// TIA Portal V20 export
DATA_BLOCK "Config"   // DB51
{ DB_Accessible_From_OPC_UA := 'FALSE' }
AUTHOR : ERsystem_FA2_DH. Kim
// stored: Access Published, DBAccessibleFromOPCUA false, DBAccessibleFromWebserver false, MemoryReserve 100, Namespace Unit1.Em5
   VAR RETAIN
      em { ExternalWritable := 'False'} : "LAF_typeEmConfiguration";
      axis { ExternalAccessible := 'False'; ExternalVisible := 'False'; ExternalWritable := 'False'} : Array[1.._.U1EM5_NO_OF_AXES] of DB_ANY;
      cam { ExternalAccessible := 'False'; ExternalVisible := 'False'; ExternalWritable := 'False'} : Array[1.._.U1EM5_NO_OF_CAM] of DB_ANY;
      outputCam { ExternalAccessible := 'False'; ExternalVisible := 'False'; ExternalWritable := 'False'} : Array[1.._.U1EM5_NO_OF_OUTPUTCAM] of DB_ANY;
      cmPnp1stCathodeDetect { S7_SetPoint := 'True'} : "LBC_typeDigitalSignalConfiguration";
      cmPnp2ndCathodeDetect { S7_SetPoint := 'True'} : "LBC_typeDigitalSignalConfiguration";
      cmCathodeAlignTableElectrodeDetect { S7_SetPoint := 'True'} : "LBC_typeDigitalSignalConfiguration";
      cmCathodeNgPnpElectrodeDetect { S7_SetPoint := 'True'} : "LBC_typeDigitalSignalConfiguration";
      cmCathodeNgBoxFullSensorDetect { S7_SetPoint := 'True'} : "LBC_typeDigitalSignalConfiguration";
      cmCathodeNgBoxDetect { S7_SetPoint := 'True'} : "LBC_typeDigitalSignalConfiguration";
      cmCathodeMainPnP1AxisX { ExternalAccessible := 'False'; ExternalVisible := 'False'; ExternalWritable := 'False'} : "LBC_typeAxis64PosConfiguration";
      cmCathodeMainPnP2AxisX { ExternalAccessible := 'False'; ExternalVisible := 'False'; ExternalWritable := 'False'} : "LBC_typeAxis64PosConfiguration";
      cmCathodeMainPnP1AxisY { ExternalAccessible := 'False'; ExternalVisible := 'False'; ExternalWritable := 'False'} : "LBC_typeAxis64PosConfiguration";
      cmCathodeMainPnP1AxisZ { ExternalAccessible := 'False'; ExternalVisible := 'False'; ExternalWritable := 'False'} : "LBC_typeAxis64PosConfiguration";
      cmCathodeMainPnP2AxisZ { ExternalAccessible := 'False'; ExternalVisible := 'False'; ExternalWritable := 'False'} : "LBC_typeAxis64PosConfiguration";
      cmCathodeAlignTableAxisX { ExternalAccessible := 'False'; ExternalVisible := 'False'; ExternalWritable := 'False'} : "LBC_typeAxis64PosConfiguration";
      cmCathodeAlignTableAxisY1 { ExternalAccessible := 'False'; ExternalVisible := 'False'; ExternalWritable := 'False'} : "LBC_typeAxis64PosConfiguration";
      cmCathodeAlignTableAxisY2 { ExternalAccessible := 'False'; ExternalVisible := 'False'; ExternalWritable := 'False'} : "LBC_typeAxis64PosConfiguration";
      cmCathodeMainPnP1RotaryCwCcw { ExternalAccessible := 'False'; ExternalVisible := 'False'; ExternalWritable := 'False'} : "LBC_typeTwoWayActuatorConfiguration";
      cmCathodeMainPnP1SuctionPlateVacuum { ExternalAccessible := 'False'; ExternalVisible := 'False'; ExternalWritable := 'False'} : "LBC_typeTwoWayActuatorConfiguration";
      cmCathodeMainPnP2SuctionPlateVacuum { ExternalAccessible := 'False'; ExternalVisible := 'False'; ExternalWritable := 'False'} : "LBC_typeTwoWayActuatorConfiguration";
      cmCathodeAlignTableSuctionPlateVacuum { ExternalAccessible := 'False'; ExternalVisible := 'False'; ExternalWritable := 'False'} : "LBC_typeTwoWayActuatorConfiguration";
      cmCathodeGlassCleaning { ExternalAccessible := 'False'; ExternalVisible := 'False'; ExternalWritable := 'False'} : "LBC_typeTwoWayActuatorConfiguration";
      cmCathodeNgPnpUpDown { ExternalAccessible := 'False'; ExternalVisible := 'False'; ExternalWritable := 'False'} : "LBC_typeTwoWayActuatorConfiguration";
      cmCathodeNgPnp1stFwdBwd { ExternalAccessible := 'False'; ExternalVisible := 'False'; ExternalWritable := 'False'; S7_SetPoint := 'True'} : "LBC_typeTwoWayActuatorConfiguration";
      cmCathodeNgPnp2ndFwdBwd { ExternalAccessible := 'False'; ExternalVisible := 'False'; ExternalWritable := 'False'; S7_SetPoint := 'True'} : "LBC_typeTwoWayActuatorConfiguration";
      cmCathodeMaintenanceMovingFixFrontRearFwdBwd { ExternalAccessible := 'False'; ExternalVisible := 'False'; ExternalWritable := 'False'} : "LBC_typeTwoWayActuatorConfiguration";
      cmCathodeNgBoxLiftUpDown { ExternalAccessible := 'False'; ExternalVisible := 'False'; ExternalWritable := 'False'; S7_SetPoint := 'True'} : "LBC_typeTwoWayActuatorConfiguration";
      cmCathodeNgBoxLockUpDown { ExternalAccessible := 'False'; ExternalVisible := 'False'; ExternalWritable := 'False'; S7_SetPoint := 'True'} : "LBC_typeTwoWayActuatorConfiguration";
      cmCathodeNgPnpVaccum { ExternalAccessible := 'False'; ExternalVisible := 'False'; ExternalWritable := 'False'; S7_SetPoint := 'True'} : "LBC_typeTwoWayActuatorConfiguration";
      cmCathodeConveyorCoverFwdBwd { S7_SetPoint := 'True'} : "LBC_typeTwoWayActuatorConfiguration";
      cmCathodeConveyorPickUpBlower { S7_SetPoint := 'True'} : "LBC_typeTwoWayActuatorConfiguration";
      cmCathodeVisionControllerInterface { ExternalAccessible := 'False'; ExternalVisible := 'False'; ExternalWritable := 'False'} : "LER_typeVisionConfiguration";
      softCam : Struct
         cmCathodeMainPnP1AxisX : "LER_typeSoftCamInterface";
         cmCathodeMainPnP2AxisX { S7_SetPoint := 'True'} : "LER_typeSoftCamInterface";
         cmCathodeMainPnP1AxisY { S7_SetPoint := 'True'} : "LER_typeSoftCamInterface";
         cmCathodeMainPnP1AxisZ { S7_SetPoint := 'True'} : "LER_typeSoftCamInterface";
         cmCathodeMainPnP2AxisZ { S7_SetPoint := 'True'} : "LER_typeSoftCamInterface";
         cmCathodeAlignTableAxisX { S7_SetPoint := 'True'} : "LER_typeSoftCamInterface";
         cmCathodeAlignTableAxisY1 { S7_SetPoint := 'True'} : "LER_typeSoftCamInterface";
         cmCathodeAlignTableAxisY2 { S7_SetPoint := 'True'} : "LER_typeSoftCamInterface";
      END_STRUCT;
   END_VAR
BEGIN
   em.referenceDesignator.parent := WSTRING#'';
   em.referenceDesignator.relative := WSTRING#'';
   em.referenceDesignator.combined := WSTRING#'';
   axis[1] := 146;   // CathodeMainPnP1AxisX
   axis[2] := 147;   // CathodeMainPnP2AxisX
   axis[3] := 152;   // CathodeMainPnP1AxisY
   axis[4] := 151;   // CathodeMainPnP1AxisZ
   axis[5] := 153;   // CathodeMainPnP2AxisZ
   axis[6] := 157;   // CathodeAlignTableAxisX
   axis[7] := 158;   // CathodeAlignTableAxisY1
   axis[8] := 159;   // CathodeAlignTableAxisY2
   cam[1] := 144;   // AnodeMainPnP1AxisX
   cam[2] := 145;   // AnodeMainPnP2AxisX
   cam[3] := 148;   // AnodeMainPnP1AxisY
   cam[4] := 149;   // AnodeMainPnP1AxisZ
   outputCam[1] := 416;
   outputCam[2] := 417;
   outputCam[3] := 419;
   outputCam[4] := 418;
   outputCam[5] := 422;
   outputCam[6] := 423;
   outputCam[7] := 428;
   outputCam[8] := 429;
   outputCam[9] := 421;
   outputCam[10] := 439;
   outputCam[11] := 427;
   outputCam[12] := 425;
   outputCam[13] := 457;
   outputCam[14] := 443;
   outputCam[15] := 424;
   outputCam[16] := 426;
   outputCam[17] := 444;
   outputCam[18] := 440;
   outputCam[19] := 458;
   cmPnp1stCathodeDetect.referenceDesignator := WSTRING#'DigitalSignal';
   cmPnp1stCathodeDetect.onDelay := T#0MS;
   cmPnp1stCathodeDetect.offDelay := T#0MS;
   cmPnp1stCathodeDetect.default := FALSE;
   cmPnp1stCathodeDetect.invertProcessValue := FALSE;
   cmPnp1stCathodeDetect.disableAlarms := FALSE;
   cmPnp2ndCathodeDetect.referenceDesignator := WSTRING#'DigitalSignal';
   cmPnp2ndCathodeDetect.onDelay := T#0MS;
   cmPnp2ndCathodeDetect.offDelay := T#0MS;
   cmPnp2ndCathodeDetect.default := FALSE;
   cmPnp2ndCathodeDetect.invertProcessValue := FALSE;
   cmPnp2ndCathodeDetect.disableAlarms := FALSE;
   cmCathodeAlignTableElectrodeDetect.referenceDesignator := WSTRING#'DigitalSignal';
   cmCathodeAlignTableElectrodeDetect.onDelay := T#0MS;
   cmCathodeAlignTableElectrodeDetect.offDelay := T#0MS;
   cmCathodeAlignTableElectrodeDetect.default := FALSE;
   cmCathodeAlignTableElectrodeDetect.invertProcessValue := FALSE;
   cmCathodeAlignTableElectrodeDetect.disableAlarms := FALSE;
   cmCathodeNgPnpElectrodeDetect.referenceDesignator := WSTRING#'DigitalSignal';
   cmCathodeNgPnpElectrodeDetect.onDelay := T#0MS;
   cmCathodeNgPnpElectrodeDetect.offDelay := T#0MS;
   cmCathodeNgPnpElectrodeDetect.default := FALSE;
   cmCathodeNgPnpElectrodeDetect.invertProcessValue := FALSE;
   cmCathodeNgPnpElectrodeDetect.disableAlarms := FALSE;
   cmCathodeNgBoxFullSensorDetect.referenceDesignator := WSTRING#'DigitalSignal';
   cmCathodeNgBoxFullSensorDetect.onDelay := T#0MS;
   cmCathodeNgBoxFullSensorDetect.offDelay := T#0MS;
   cmCathodeNgBoxFullSensorDetect.default := FALSE;
   cmCathodeNgBoxFullSensorDetect.invertProcessValue := FALSE;
   cmCathodeNgBoxFullSensorDetect.disableAlarms := FALSE;
   cmCathodeNgBoxDetect.referenceDesignator := WSTRING#'DigitalSignal';
   cmCathodeNgBoxDetect.onDelay := T#0MS;
   cmCathodeNgBoxDetect.offDelay := T#0MS;
   cmCathodeNgBoxDetect.default := FALSE;
   cmCathodeNgBoxDetect.invertProcessValue := FALSE;
   cmCathodeNgBoxDetect.disableAlarms := FALSE;
   cmCathodeMainPnP1AxisX.referenceDesignator := WSTRING#'CathodeMainPnP1AxisX';
   cmCathodeMainPnP1AxisX.disableAlarms := FALSE;
   cmCathodeMainPnP1AxisX.masterControlPopUp := TRUE;
   cmCathodeMainPnP1AxisX.setPositions[0].position := 0.0;
   cmCathodeMainPnP1AxisX.setPositions[1].position := 540.0;
   cmCathodeMainPnP1AxisX.setPositions[2].position := 544.0;
   cmCathodeMainPnP1AxisX.setPositions[3..15].position := 0.0;
   cmCathodeMainPnP1AxisX.setPositions[0..1].velocity := 500.0;
   cmCathodeMainPnP1AxisX.setPositions[2..3].velocity := 1040.0;
   cmCathodeMainPnP1AxisX.setPositions[4..15].velocity := -1.0;
   cmCathodeMainPnP1AxisX.setPositions[0..1].acceleration := 5000.0;
   cmCathodeMainPnP1AxisX.setPositions[2..3].acceleration := 10400.0;
   cmCathodeMainPnP1AxisX.setPositions[4..15].acceleration := -1.0;
   cmCathodeMainPnP1AxisX.setPositions[0..1].deceleration := 5000.0;
   cmCathodeMainPnP1AxisX.setPositions[2..3].deceleration := 10400.0;
   cmCathodeMainPnP1AxisX.setPositions[4..15].deceleration := -1.0;
   cmCathodeMainPnP1AxisX.setPositions[0..15]."name" := '';
   cmCathodeMainPnP2AxisX.referenceDesignator := WSTRING#'CathodeMainPnP2AxisX';
   cmCathodeMainPnP2AxisX.disableAlarms := FALSE;
   cmCathodeMainPnP2AxisX.masterControlPopUp := TRUE;
   cmCathodeMainPnP2AxisX.setPositions[0].position := 0.0;
   cmCathodeMainPnP2AxisX.setPositions[1].position := 540.0;
   cmCathodeMainPnP2AxisX.setPositions[2].position := 538.0;
   cmCathodeMainPnP2AxisX.setPositions[3..15].position := 0.0;
   cmCathodeMainPnP2AxisX.setPositions[0..1].velocity := 500.0;
   cmCathodeMainPnP2AxisX.setPositions[2..3].velocity := 1040.0;
   cmCathodeMainPnP2AxisX.setPositions[4..15].velocity := -1.0;
   cmCathodeMainPnP2AxisX.setPositions[0..1].acceleration := 5000.0;
   cmCathodeMainPnP2AxisX.setPositions[2..3].acceleration := 10400.0;
   cmCathodeMainPnP2AxisX.setPositions[4..15].acceleration := -1.0;
   cmCathodeMainPnP2AxisX.setPositions[0..1].deceleration := 5000.0;
   cmCathodeMainPnP2AxisX.setPositions[2..3].deceleration := 10400.0;
   cmCathodeMainPnP2AxisX.setPositions[4..15].deceleration := -1.0;
   cmCathodeMainPnP2AxisX.setPositions[0..15]."name" := '';
   cmCathodeMainPnP1AxisY.referenceDesignator := WSTRING#'CathodeMainPnP1AxisY';
   cmCathodeMainPnP1AxisY.disableAlarms := FALSE;
   cmCathodeMainPnP1AxisY.masterControlPopUp := TRUE;
   cmCathodeMainPnP1AxisY.setPositions[0..15].position := 0.0;
   cmCathodeMainPnP1AxisY.setPositions[0].velocity := 50.0;
   cmCathodeMainPnP1AxisY.setPositions[1].velocity := 30.0;
   cmCathodeMainPnP1AxisY.setPositions[2..15].velocity := -1.0;
   cmCathodeMainPnP1AxisY.setPositions[0].acceleration := 500.0;
   cmCathodeMainPnP1AxisY.setPositions[1].acceleration := 30.0;
   cmCathodeMainPnP1AxisY.setPositions[2..15].acceleration := -1.0;
   cmCathodeMainPnP1AxisY.setPositions[0].deceleration := 500.0;
   cmCathodeMainPnP1AxisY.setPositions[1].deceleration := 30.0;
   cmCathodeMainPnP1AxisY.setPositions[2..15].deceleration := -1.0;
   cmCathodeMainPnP1AxisY.setPositions[0..15]."name" := '';
   cmCathodeMainPnP1AxisZ.referenceDesignator := WSTRING#'CathodeMainPnP1AxisZ';
   cmCathodeMainPnP1AxisZ.disableAlarms := FALSE;
   cmCathodeMainPnP1AxisZ.masterControlPopUp := TRUE;
   cmCathodeMainPnP1AxisZ.setPositions[0].position := 0.0;
   cmCathodeMainPnP1AxisZ.setPositions[1].position := 20.0;
   cmCathodeMainPnP1AxisZ.setPositions[2].position := 30.0;
   cmCathodeMainPnP1AxisZ.setPositions[3..15].position := 0.0;
   cmCathodeMainPnP1AxisZ.setPositions[0..3].velocity := 50.0;
   cmCathodeMainPnP1AxisZ.setPositions[4..15].velocity := -1.0;
   cmCathodeMainPnP1AxisZ.setPositions[0..3].acceleration := 500.0;
   cmCathodeMainPnP1AxisZ.setPositions[4..15].acceleration := -1.0;
   cmCathodeMainPnP1AxisZ.setPositions[0..3].deceleration := 500.0;
   cmCathodeMainPnP1AxisZ.setPositions[4..15].deceleration := -1.0;
   cmCathodeMainPnP1AxisZ.setPositions[0..15]."name" := '';
   cmCathodeMainPnP2AxisZ.referenceDesignator := WSTRING#'CathodeMainPnP2AxisZ';
   cmCathodeMainPnP2AxisZ.disableAlarms := FALSE;
   cmCathodeMainPnP2AxisZ.masterControlPopUp := TRUE;
   cmCathodeMainPnP2AxisZ.setPositions[0].position := 0.0;
   cmCathodeMainPnP2AxisZ.setPositions[1].position := 20.0;
   cmCathodeMainPnP2AxisZ.setPositions[2].position := 30.0;
   cmCathodeMainPnP2AxisZ.setPositions[3..15].position := 0.0;
   cmCathodeMainPnP2AxisZ.setPositions[0..3].velocity := 50.0;
   cmCathodeMainPnP2AxisZ.setPositions[4..15].velocity := -1.0;
   cmCathodeMainPnP2AxisZ.setPositions[0..3].acceleration := 500.0;
   cmCathodeMainPnP2AxisZ.setPositions[4..15].acceleration := -1.0;
   cmCathodeMainPnP2AxisZ.setPositions[0..3].deceleration := 500.0;
   cmCathodeMainPnP2AxisZ.setPositions[4..15].deceleration := -1.0;
   cmCathodeMainPnP2AxisZ.setPositions[0..15]."name" := '';
   cmCathodeAlignTableAxisX.referenceDesignator := WSTRING#'CathodeAlignTableAxisX';
   cmCathodeAlignTableAxisX.disableAlarms := FALSE;
   cmCathodeAlignTableAxisX.masterControlPopUp := TRUE;
   cmCathodeAlignTableAxisX.setPositions[0].position := 0.0;
   cmCathodeAlignTableAxisX.setPositions[1].position := 1.0;
   cmCathodeAlignTableAxisX.setPositions[2..3].position := 1.07;
   cmCathodeAlignTableAxisX.setPositions[4].position := -0.93;
   cmCathodeAlignTableAxisX.setPositions[5..7].position := -2.93;
   cmCathodeAlignTableAxisX.setPositions[8].position := -0.93;
   cmCathodeAlignTableAxisX.setPositions[9].position := 1.07;
   cmCathodeAlignTableAxisX.setPositions[10..15].position := 0.0;
   cmCathodeAlignTableAxisX.setPositions[0..1].velocity := 50.0;
   cmCathodeAlignTableAxisX.setPositions[2..9].velocity := 30.0;
   cmCathodeAlignTableAxisX.setPositions[10..15].velocity := -1.0;
   cmCathodeAlignTableAxisX.setPositions[0..1].acceleration := 500.0;
   cmCathodeAlignTableAxisX.setPositions[2..9].acceleration := 30.0;
   cmCathodeAlignTableAxisX.setPositions[10..15].acceleration := -1.0;
   cmCathodeAlignTableAxisX.setPositions[0..1].deceleration := 500.0;
   cmCathodeAlignTableAxisX.setPositions[2..9].deceleration := 30.0;
   cmCathodeAlignTableAxisX.setPositions[10..15].deceleration := -1.0;
   cmCathodeAlignTableAxisX.setPositions[0..15]."name" := '';
   cmCathodeAlignTableAxisY1.referenceDesignator := WSTRING#'CathodeAlignTableAxisY1';
   cmCathodeAlignTableAxisY1.disableAlarms := FALSE;
   cmCathodeAlignTableAxisY1.masterControlPopUp := TRUE;
   cmCathodeAlignTableAxisY1.setPositions[0].position := 0.0;
   cmCathodeAlignTableAxisY1.setPositions[1].position := 2.0;
   cmCathodeAlignTableAxisY1.setPositions[2].position := 0.15;
   cmCathodeAlignTableAxisY1.setPositions[3..5].position := 2.15;
   cmCathodeAlignTableAxisY1.setPositions[6].position := 0.15;
   cmCathodeAlignTableAxisY1.setPositions[7].position := -1.85;
   cmCathodeAlignTableAxisY1.setPositions[8].position := 0.15;
   cmCathodeAlignTableAxisY1.setPositions[9].position := -1.85;
   cmCathodeAlignTableAxisY1.setPositions[10..15].position := 0.0;
   cmCathodeAlignTableAxisY1.setPositions[0..1].velocity := 50.0;
   cmCathodeAlignTableAxisY1.setPositions[2..9].velocity := 30.0;
   cmCathodeAlignTableAxisY1.setPositions[10..15].velocity := -1.0;
   cmCathodeAlignTableAxisY1.setPositions[0..1].acceleration := 500.0;
   cmCathodeAlignTableAxisY1.setPositions[2..9].acceleration := 30.0;
   cmCathodeAlignTableAxisY1.setPositions[10..15].acceleration := -1.0;
   cmCathodeAlignTableAxisY1.setPositions[0..1].deceleration := 500.0;
   cmCathodeAlignTableAxisY1.setPositions[2..9].deceleration := 30.0;
   cmCathodeAlignTableAxisY1.setPositions[10..15].deceleration := -1.0;
   cmCathodeAlignTableAxisY1.setPositions[0..15]."name" := '';
   cmCathodeAlignTableAxisY2.referenceDesignator := WSTRING#'CathodeAlignTableAxisY2';
   cmCathodeAlignTableAxisY2.disableAlarms := FALSE;
   cmCathodeAlignTableAxisY2.masterControlPopUp := TRUE;
   cmCathodeAlignTableAxisY2.setPositions[0].position := 0.0;
   cmCathodeAlignTableAxisY2.setPositions[1].position := 3.0;
   cmCathodeAlignTableAxisY2.setPositions[2].position := -0.96;
   cmCathodeAlignTableAxisY2.setPositions[3..5].position := -2.96;
   cmCathodeAlignTableAxisY2.setPositions[6].position := -0.96;
   cmCathodeAlignTableAxisY2.setPositions[7].position := 1.04;
   cmCathodeAlignTableAxisY2.setPositions[8].position := -0.96;
   cmCathodeAlignTableAxisY2.setPositions[9].position := 1.04;
   cmCathodeAlignTableAxisY2.setPositions[10..15].position := 0.0;
   cmCathodeAlignTableAxisY2.setPositions[0..1].velocity := 50.0;
   cmCathodeAlignTableAxisY2.setPositions[2..9].velocity := 30.0;
   cmCathodeAlignTableAxisY2.setPositions[10..15].velocity := -1.0;
   cmCathodeAlignTableAxisY2.setPositions[0..1].acceleration := 500.0;
   cmCathodeAlignTableAxisY2.setPositions[2..9].acceleration := 30.0;
   cmCathodeAlignTableAxisY2.setPositions[10..15].acceleration := -1.0;
   cmCathodeAlignTableAxisY2.setPositions[0..1].deceleration := 500.0;
   cmCathodeAlignTableAxisY2.setPositions[2..9].deceleration := 30.0;
   cmCathodeAlignTableAxisY2.setPositions[10..15].deceleration := -1.0;
   cmCathodeAlignTableAxisY2.setPositions[0..15]."name" := '';
   cmCathodeMainPnP1RotaryCwCcw.referenceDesignator := WSTRING#'MainPnP1RotaryCwCcw';
   cmCathodeMainPnP1RotaryCwCcw.monitoringLeavingFeedback := T#1S;
   cmCathodeMainPnP1RotaryCwCcw.monitoringReachingFeedback := T#1S;
   cmCathodeMainPnP1RotaryCwCcw.monitoringDiscrepancy := T#0MS;
   cmCathodeMainPnP1RotaryCwCcw.setOutputHomeContinuously := TRUE;
   cmCathodeMainPnP1RotaryCwCcw.setOutputWorkContinuously := TRUE;
   cmCathodeMainPnP1RotaryCwCcw.disableHomeCommand := FALSE;
   cmCathodeMainPnP1RotaryCwCcw.disableFeedbackHomePos := FALSE;
   cmCathodeMainPnP1RotaryCwCcw.disableFeedbackWorkPos := FALSE;
   cmCathodeMainPnP1RotaryCwCcw.disableAlarms := TRUE;
   cmCathodeMainPnP1RotaryCwCcw.resetOutputsOnError := FALSE;
   cmCathodeMainPnP1RotaryCwCcw.allwaysWaitOnReachingTime := FALSE;
   cmCathodeMainPnP1SuctionPlateVacuum.referenceDesignator := WSTRING#'MainPnP1Vacuum';
   cmCathodeMainPnP1SuctionPlateVacuum.monitoringLeavingFeedback := T#1S;
   cmCathodeMainPnP1SuctionPlateVacuum.monitoringReachingFeedback := T#1S;
   cmCathodeMainPnP1SuctionPlateVacuum.monitoringDiscrepancy := T#15S;
   cmCathodeMainPnP1SuctionPlateVacuum.setOutputHomeContinuously := TRUE;
   cmCathodeMainPnP1SuctionPlateVacuum.setOutputWorkContinuously := TRUE;
   cmCathodeMainPnP1SuctionPlateVacuum.disableHomeCommand := FALSE;
   cmCathodeMainPnP1SuctionPlateVacuum.disableFeedbackHomePos := FALSE;
   cmCathodeMainPnP1SuctionPlateVacuum.disableFeedbackWorkPos := FALSE;
   cmCathodeMainPnP1SuctionPlateVacuum.disableAlarms := FALSE;
   cmCathodeMainPnP1SuctionPlateVacuum.resetOutputsOnError := FALSE;
   cmCathodeMainPnP1SuctionPlateVacuum.allwaysWaitOnReachingTime := FALSE;
   cmCathodeMainPnP2SuctionPlateVacuum.referenceDesignator := WSTRING#'MainPnP2Vacuum';
   cmCathodeMainPnP2SuctionPlateVacuum.monitoringLeavingFeedback := T#1S;
   cmCathodeMainPnP2SuctionPlateVacuum.monitoringReachingFeedback := T#1S;
   cmCathodeMainPnP2SuctionPlateVacuum.monitoringDiscrepancy := T#15S;
   cmCathodeMainPnP2SuctionPlateVacuum.setOutputHomeContinuously := TRUE;
   cmCathodeMainPnP2SuctionPlateVacuum.setOutputWorkContinuously := TRUE;
   cmCathodeMainPnP2SuctionPlateVacuum.disableHomeCommand := FALSE;
   cmCathodeMainPnP2SuctionPlateVacuum.disableFeedbackHomePos := FALSE;
   cmCathodeMainPnP2SuctionPlateVacuum.disableFeedbackWorkPos := FALSE;
   cmCathodeMainPnP2SuctionPlateVacuum.disableAlarms := FALSE;
   cmCathodeMainPnP2SuctionPlateVacuum.resetOutputsOnError := FALSE;
   cmCathodeMainPnP2SuctionPlateVacuum.allwaysWaitOnReachingTime := FALSE;
   cmCathodeAlignTableSuctionPlateVacuum.referenceDesignator := WSTRING#'AlignTableVaccum';
   cmCathodeAlignTableSuctionPlateVacuum.monitoringLeavingFeedback := T#1S;
   cmCathodeAlignTableSuctionPlateVacuum.monitoringReachingFeedback := T#1S;
   cmCathodeAlignTableSuctionPlateVacuum.monitoringDiscrepancy := T#0MS;
   cmCathodeAlignTableSuctionPlateVacuum.setOutputHomeContinuously := TRUE;
   cmCathodeAlignTableSuctionPlateVacuum.setOutputWorkContinuously := TRUE;
   cmCathodeAlignTableSuctionPlateVacuum.disableHomeCommand := FALSE;
   cmCathodeAlignTableSuctionPlateVacuum.disableFeedbackHomePos := FALSE;
   cmCathodeAlignTableSuctionPlateVacuum.disableFeedbackWorkPos := FALSE;
   cmCathodeAlignTableSuctionPlateVacuum.disableAlarms := FALSE;
   cmCathodeAlignTableSuctionPlateVacuum.resetOutputsOnError := FALSE;
   cmCathodeAlignTableSuctionPlateVacuum.allwaysWaitOnReachingTime := FALSE;
   cmCathodeGlassCleaning.referenceDesignator := WSTRING#'GlassCleaning';
   cmCathodeGlassCleaning.monitoringLeavingFeedback := T#1S;
   cmCathodeGlassCleaning.monitoringReachingFeedback := T#1S;
   cmCathodeGlassCleaning.monitoringDiscrepancy := T#0MS;
   cmCathodeGlassCleaning.setOutputHomeContinuously := TRUE;
   cmCathodeGlassCleaning.setOutputWorkContinuously := TRUE;
   cmCathodeGlassCleaning.disableHomeCommand := FALSE;
   cmCathodeGlassCleaning.disableFeedbackHomePos := TRUE;
   cmCathodeGlassCleaning.disableFeedbackWorkPos := TRUE;
   cmCathodeGlassCleaning.disableAlarms := TRUE;
   cmCathodeGlassCleaning.resetOutputsOnError := FALSE;
   cmCathodeGlassCleaning.allwaysWaitOnReachingTime := FALSE;
   cmCathodeNgPnpUpDown.referenceDesignator := WSTRING#'NgPnpUpDown';
   cmCathodeNgPnpUpDown.monitoringLeavingFeedback := T#5S;
   cmCathodeNgPnpUpDown.monitoringReachingFeedback := T#5S;
   cmCathodeNgPnpUpDown.monitoringDiscrepancy := T#0MS;
   cmCathodeNgPnpUpDown.setOutputHomeContinuously := TRUE;
   cmCathodeNgPnpUpDown.setOutputWorkContinuously := TRUE;
   cmCathodeNgPnpUpDown.disableHomeCommand := FALSE;
   cmCathodeNgPnpUpDown.disableFeedbackHomePos := TRUE;
   cmCathodeNgPnpUpDown.disableFeedbackWorkPos := TRUE;
   cmCathodeNgPnpUpDown.disableAlarms := FALSE;
   cmCathodeNgPnpUpDown.resetOutputsOnError := FALSE;
   cmCathodeNgPnpUpDown.allwaysWaitOnReachingTime := FALSE;
   cmCathodeNgPnp1stFwdBwd.referenceDesignator := WSTRING#'NgPnp1stFwdBwd';
   cmCathodeNgPnp1stFwdBwd.monitoringLeavingFeedback := T#5S;
   cmCathodeNgPnp1stFwdBwd.monitoringReachingFeedback := T#5S;
   cmCathodeNgPnp1stFwdBwd.monitoringDiscrepancy := T#0MS;
   cmCathodeNgPnp1stFwdBwd.setOutputHomeContinuously := TRUE;
   cmCathodeNgPnp1stFwdBwd.setOutputWorkContinuously := TRUE;
   cmCathodeNgPnp1stFwdBwd.disableHomeCommand := FALSE;
   cmCathodeNgPnp1stFwdBwd.disableFeedbackHomePos := FALSE;
   cmCathodeNgPnp1stFwdBwd.disableFeedbackWorkPos := FALSE;
   cmCathodeNgPnp1stFwdBwd.disableAlarms := FALSE;
   cmCathodeNgPnp1stFwdBwd.resetOutputsOnError := FALSE;
   cmCathodeNgPnp1stFwdBwd.allwaysWaitOnReachingTime := FALSE;
   cmCathodeNgPnp2ndFwdBwd.referenceDesignator := WSTRING#'NgPnp2ndFwdBwd';
   cmCathodeNgPnp2ndFwdBwd.monitoringLeavingFeedback := T#5S;
   cmCathodeNgPnp2ndFwdBwd.monitoringReachingFeedback := T#5S;
   cmCathodeNgPnp2ndFwdBwd.monitoringDiscrepancy := T#0MS;
   cmCathodeNgPnp2ndFwdBwd.setOutputHomeContinuously := TRUE;
   cmCathodeNgPnp2ndFwdBwd.setOutputWorkContinuously := TRUE;
   cmCathodeNgPnp2ndFwdBwd.disableHomeCommand := FALSE;
   cmCathodeNgPnp2ndFwdBwd.disableFeedbackHomePos := TRUE;
   cmCathodeNgPnp2ndFwdBwd.disableFeedbackWorkPos := TRUE;
   cmCathodeNgPnp2ndFwdBwd.disableAlarms := FALSE;
   cmCathodeNgPnp2ndFwdBwd.resetOutputsOnError := FALSE;
   cmCathodeNgPnp2ndFwdBwd.allwaysWaitOnReachingTime := FALSE;
   cmCathodeMaintenanceMovingFixFrontRearFwdBwd.referenceDesignator := WSTRING#'MaintenanceFix';
   cmCathodeMaintenanceMovingFixFrontRearFwdBwd.monitoringLeavingFeedback := T#5S;
   cmCathodeMaintenanceMovingFixFrontRearFwdBwd.monitoringReachingFeedback := T#5S;
   cmCathodeMaintenanceMovingFixFrontRearFwdBwd.monitoringDiscrepancy := T#0MS;
   cmCathodeMaintenanceMovingFixFrontRearFwdBwd.setOutputHomeContinuously := TRUE;
   cmCathodeMaintenanceMovingFixFrontRearFwdBwd.setOutputWorkContinuously := TRUE;
   cmCathodeMaintenanceMovingFixFrontRearFwdBwd.disableHomeCommand := FALSE;
   cmCathodeMaintenanceMovingFixFrontRearFwdBwd.disableFeedbackHomePos := FALSE;
   cmCathodeMaintenanceMovingFixFrontRearFwdBwd.disableFeedbackWorkPos := FALSE;
   cmCathodeMaintenanceMovingFixFrontRearFwdBwd.disableAlarms := FALSE;
   cmCathodeMaintenanceMovingFixFrontRearFwdBwd.resetOutputsOnError := FALSE;
   cmCathodeMaintenanceMovingFixFrontRearFwdBwd.allwaysWaitOnReachingTime := FALSE;
   cmCathodeNgBoxLiftUpDown.referenceDesignator := WSTRING#'NgBoxLiftUpDown';
   cmCathodeNgBoxLiftUpDown.monitoringLeavingFeedback := T#5S;
   cmCathodeNgBoxLiftUpDown.monitoringReachingFeedback := T#5S;
   cmCathodeNgBoxLiftUpDown.monitoringDiscrepancy := T#0MS;
   cmCathodeNgBoxLiftUpDown.setOutputHomeContinuously := TRUE;
   cmCathodeNgBoxLiftUpDown.setOutputWorkContinuously := TRUE;
   cmCathodeNgBoxLiftUpDown.disableHomeCommand := FALSE;
   cmCathodeNgBoxLiftUpDown.disableFeedbackHomePos := FALSE;
   cmCathodeNgBoxLiftUpDown.disableFeedbackWorkPos := FALSE;
   cmCathodeNgBoxLiftUpDown.disableAlarms := FALSE;
   cmCathodeNgBoxLiftUpDown.resetOutputsOnError := FALSE;
   cmCathodeNgBoxLiftUpDown.allwaysWaitOnReachingTime := FALSE;
   cmCathodeNgBoxLockUpDown.referenceDesignator := WSTRING#'NgBoxLockUpDown';
   cmCathodeNgBoxLockUpDown.monitoringLeavingFeedback := T#5S;
   cmCathodeNgBoxLockUpDown.monitoringReachingFeedback := T#5S;
   cmCathodeNgBoxLockUpDown.monitoringDiscrepancy := T#0MS;
   cmCathodeNgBoxLockUpDown.setOutputHomeContinuously := TRUE;
   cmCathodeNgBoxLockUpDown.setOutputWorkContinuously := TRUE;
   cmCathodeNgBoxLockUpDown.disableHomeCommand := FALSE;
   cmCathodeNgBoxLockUpDown.disableFeedbackHomePos := FALSE;
   cmCathodeNgBoxLockUpDown.disableFeedbackWorkPos := FALSE;
   cmCathodeNgBoxLockUpDown.disableAlarms := FALSE;
   cmCathodeNgBoxLockUpDown.resetOutputsOnError := FALSE;
   cmCathodeNgBoxLockUpDown.allwaysWaitOnReachingTime := FALSE;
   cmCathodeNgPnpVaccum.referenceDesignator := WSTRING#'NgPnpVaccum';
   cmCathodeNgPnpVaccum.monitoringLeavingFeedback := T#5S;
   cmCathodeNgPnpVaccum.monitoringReachingFeedback := T#5S;
   cmCathodeNgPnpVaccum.monitoringDiscrepancy := T#0MS;
   cmCathodeNgPnpVaccum.setOutputHomeContinuously := TRUE;
   cmCathodeNgPnpVaccum.setOutputWorkContinuously := TRUE;
   cmCathodeNgPnpVaccum.disableHomeCommand := FALSE;
   cmCathodeNgPnpVaccum.disableFeedbackHomePos := FALSE;
   cmCathodeNgPnpVaccum.disableFeedbackWorkPos := FALSE;
   cmCathodeNgPnpVaccum.disableAlarms := FALSE;
   cmCathodeNgPnpVaccum.resetOutputsOnError := FALSE;
   cmCathodeNgPnpVaccum.allwaysWaitOnReachingTime := FALSE;
   cmCathodeConveyorCoverFwdBwd.referenceDesignator := WSTRING#'ConveyorCoverFwdBwd';
   cmCathodeConveyorCoverFwdBwd.monitoringLeavingFeedback := T#5S;
   cmCathodeConveyorCoverFwdBwd.monitoringReachingFeedback := T#5S;
   cmCathodeConveyorCoverFwdBwd.monitoringDiscrepancy := T#0MS;
   cmCathodeConveyorCoverFwdBwd.setOutputHomeContinuously := TRUE;
   cmCathodeConveyorCoverFwdBwd.setOutputWorkContinuously := TRUE;
   cmCathodeConveyorCoverFwdBwd.disableHomeCommand := FALSE;
   cmCathodeConveyorCoverFwdBwd.disableFeedbackHomePos := TRUE;
   cmCathodeConveyorCoverFwdBwd.disableFeedbackWorkPos := TRUE;
   cmCathodeConveyorCoverFwdBwd.disableAlarms := FALSE;
   cmCathodeConveyorCoverFwdBwd.resetOutputsOnError := FALSE;
   cmCathodeConveyorCoverFwdBwd.allwaysWaitOnReachingTime := FALSE;
   cmCathodeConveyorPickUpBlower.referenceDesignator := WSTRING#'ConveyorPickUpBlower';
   cmCathodeConveyorPickUpBlower.monitoringLeavingFeedback := T#0MS;
   cmCathodeConveyorPickUpBlower.monitoringReachingFeedback := T#0MS;
   cmCathodeConveyorPickUpBlower.monitoringDiscrepancy := T#0MS;
   cmCathodeConveyorPickUpBlower.setOutputHomeContinuously := TRUE;
   cmCathodeConveyorPickUpBlower.setOutputWorkContinuously := TRUE;
   cmCathodeConveyorPickUpBlower.disableHomeCommand := FALSE;
   cmCathodeConveyorPickUpBlower.disableFeedbackHomePos := TRUE;
   cmCathodeConveyorPickUpBlower.disableFeedbackWorkPos := TRUE;
   cmCathodeConveyorPickUpBlower.disableAlarms := FALSE;
   cmCathodeConveyorPickUpBlower.resetOutputsOnError := FALSE;
   cmCathodeConveyorPickUpBlower.allwaysWaitOnReachingTime := FALSE;
   cmCathodeVisionControllerInterface.hwID.cmdResultStatusID := 770;
   cmCathodeVisionControllerInterface.hwID.trgReadyStatusID := 771;
   cmCathodeVisionControllerInterface.hwID.trgAckStatusID := 772;
   cmCathodeVisionControllerInterface.hwID.miscellaneousStatusID := 773;
   cmCathodeVisionControllerInterface.hwID.assignableStatusID := 774;
   cmCathodeVisionControllerInterface.hwID.resultData248ByteID_1 := 791;
   cmCathodeVisionControllerInterface.hwID.resultData248ByteID_2 := 984;
   cmCathodeVisionControllerInterface.hwID.resultData248ByteID_3 := 987;
   cmCathodeVisionControllerInterface.hwID.resultData248ByteID_4 := 988;
   cmCathodeVisionControllerInterface.hwID.resultData248ByteID_5 := 989;
   cmCathodeVisionControllerInterface.hwID.cmdResultControlID := 940;
   cmCathodeVisionControllerInterface.hwID.trgControlID := 941;
   cmCathodeVisionControllerInterface.hwID.miscellaneousControlID := 942;
   cmCathodeVisionControllerInterface.hwID.reservedControlID := 943;
   cmCathodeVisionControllerInterface.hwID.assignableControlID := 944;
   cmCathodeVisionControllerInterface.hwID.parameterData248ByteID_1 := 945;
   cmCathodeVisionControllerInterface.hwID.parameterData248ByteID_2 := 990;
   cmCathodeVisionControllerInterface.hwID.parameterData248ByteID_3 := 991;
   cmCathodeVisionControllerInterface.hwID.parameterData248ByteID_4 := 992;
   cmCathodeVisionControllerInterface.hwID.parameterData248ByteID_5 := 993;
   cmCathodeVisionControllerInterface.referenceDesignator := WSTRING#'';
   cmCathodeVisionControllerInterface.disableAlarms := FALSE;
   cmCathodeVisionControllerInterface.trigger1Use := FALSE;
   cmCathodeVisionControllerInterface.trigger2Use := FALSE;
   cmCathodeVisionControllerInterface.trigger3Use := FALSE;
   cmCathodeVisionControllerInterface.trigger4Use := FALSE;
   cmCathodeVisionControllerInterface.triggertime := T#0MS;
   cmCathodeVisionControllerInterface.cycleTime := T#0MS;
   cmCathodeVisionControllerInterface.DataConfig.cmdResultControl.cmdRequest := FALSE;
   cmCathodeVisionControllerInterface.DataConfig.cmdResultControl.inDataFbSyncInhibit := FALSE;
   cmCathodeVisionControllerInterface.DataConfig.cmdResultControl.reserved := FALSE;
   cmCathodeVisionControllerInterface.DataConfig.cmdResultControl.resultAck := FALSE;
   cmCathodeVisionControllerInterface.DataConfig.cmdResultControl.err0ResetRequest := FALSE;
   cmCathodeVisionControllerInterface.DataConfig.cmdResultControl.err1ResetRequest := FALSE;
   cmCathodeVisionControllerInterface.DataConfig.cmdResultControl.reserved0 := FALSE;
   cmCathodeVisionControllerInterface.DataConfig.cmdResultControl.reserved1 := FALSE;
   cmCathodeVisionControllerInterface.DataConfig.trgControl.trg1 := FALSE;
   cmCathodeVisionControllerInterface.DataConfig.trgControl.trg2 := FALSE;
   cmCathodeVisionControllerInterface.DataConfig.trgControl.trg3 := FALSE;
   cmCathodeVisionControllerInterface.DataConfig.trgControl.trg4 := FALSE;
   cmCathodeVisionControllerInterface.DataConfig.trgControl.reserved0 := FALSE;
   cmCathodeVisionControllerInterface.DataConfig.trgControl.reserved1 := FALSE;
   cmCathodeVisionControllerInterface.DataConfig.trgControl.reserved2 := FALSE;
   cmCathodeVisionControllerInterface.DataConfig.trgControl.reserved3 := FALSE;
   cmCathodeVisionControllerInterface.DataConfig.miscellaneousControl.reset := FALSE;
   cmCathodeVisionControllerInterface.DataConfig.miscellaneousControl.ext := FALSE;
   cmCathodeVisionControllerInterface.DataConfig.miscellaneousControl.test := FALSE;
   cmCathodeVisionControllerInterface.DataConfig.miscellaneousControl.reserved0 := FALSE;
   cmCathodeVisionControllerInterface.DataConfig.miscellaneousControl.reserved1 := FALSE;
   cmCathodeVisionControllerInterface.DataConfig.miscellaneousControl.reserved2 := FALSE;
   cmCathodeVisionControllerInterface.DataConfig.miscellaneousControl.reserved3 := FALSE;
   cmCathodeVisionControllerInterface.DataConfig.miscellaneousControl.reserved4 := FALSE;
   cmCathodeVisionControllerInterface.DataConfig.reservedControl.reserved0 := FALSE;
   cmCathodeVisionControllerInterface.DataConfig.reservedControl.reserved1 := FALSE;
   cmCathodeVisionControllerInterface.DataConfig.reservedControl.reserved2 := FALSE;
   cmCathodeVisionControllerInterface.DataConfig.reservedControl.reserved3 := FALSE;
   cmCathodeVisionControllerInterface.DataConfig.reservedControl.reserved4 := FALSE;
   cmCathodeVisionControllerInterface.DataConfig.reservedControl.reserved5 := FALSE;
   cmCathodeVisionControllerInterface.DataConfig.reservedControl.reserved6 := FALSE;
   cmCathodeVisionControllerInterface.DataConfig.reservedControl.reserved7 := FALSE;
   cmCathodeVisionControllerInterface.DataConfig.assignableControl.assignable_0 := FALSE;
   cmCathodeVisionControllerInterface.DataConfig.assignableControl.assignable_1 := FALSE;
   cmCathodeVisionControllerInterface.DataConfig.assignableControl.assignable_2 := FALSE;
   cmCathodeVisionControllerInterface.DataConfig.assignableControl.assignable_3 := FALSE;
   cmCathodeVisionControllerInterface.DataConfig.assignableControl.assignable_4 := FALSE;
   cmCathodeVisionControllerInterface.DataConfig.assignableControl.assignable_5 := FALSE;
   cmCathodeVisionControllerInterface.DataConfig.assignableControl.assignable_6 := FALSE;
   cmCathodeVisionControllerInterface.DataConfig.assignableControl.assignable_7 := FALSE;
   cmCathodeVisionControllerInterface.DataConfig.assignableControl.assignable_8 := FALSE;
   cmCathodeVisionControllerInterface.DataConfig.assignableControl.assignable_9 := FALSE;
   cmCathodeVisionControllerInterface.DataConfig.assignableControl.assignable_10 := FALSE;
   cmCathodeVisionControllerInterface.DataConfig.assignableControl.assignable_11 := FALSE;
   cmCathodeVisionControllerInterface.DataConfig.assignableControl.assignable_12 := FALSE;
   cmCathodeVisionControllerInterface.DataConfig.assignableControl.assignable_13 := FALSE;
   cmCathodeVisionControllerInterface.DataConfig.assignableControl.assignable_14 := FALSE;
   cmCathodeVisionControllerInterface.DataConfig.assignableControl.assignable_15 := FALSE;
   cmCathodeVisionControllerInterface.DataConfig.assignableControl.assignable_16 := FALSE;
   cmCathodeVisionControllerInterface.DataConfig.assignableControl.assignable_17 := FALSE;
   cmCathodeVisionControllerInterface.DataConfig.assignableControl.assignable_18 := FALSE;
   cmCathodeVisionControllerInterface.DataConfig.assignableControl.assignable_19 := FALSE;
   cmCathodeVisionControllerInterface.DataConfig.assignableControl.assignable_20 := FALSE;
   cmCathodeVisionControllerInterface.DataConfig.assignableControl.assignable_21 := FALSE;
   cmCathodeVisionControllerInterface.DataConfig.assignableControl.assignable_22 := FALSE;
   cmCathodeVisionControllerInterface.DataConfig.assignableControl.assignable_23 := FALSE;
   cmCathodeVisionControllerInterface.DataConfig.assignableControl.assignable_24 := FALSE;
   cmCathodeVisionControllerInterface.DataConfig.assignableControl.assignable_25 := FALSE;
   cmCathodeVisionControllerInterface.DataConfig.assignableControl.assignable_26 := FALSE;
   cmCathodeVisionControllerInterface.DataConfig.assignableControl.assignable_27 := FALSE;
   cmCathodeVisionControllerInterface.DataConfig.assignableControl.assignable_28 := FALSE;
   cmCathodeVisionControllerInterface.DataConfig.assignableControl.assignable_29 := FALSE;
   cmCathodeVisionControllerInterface.DataConfig.assignableControl.assignable_30 := FALSE;
   cmCathodeVisionControllerInterface.DataConfig.assignableControl.assignable_31 := FALSE;
   cmCathodeVisionControllerInterface.DataConfig.parameterData248Byte_1.reversed0 := 0;
   cmCathodeVisionControllerInterface.DataConfig.parameterData248Byte_1.reserved1 := 0;
   cmCathodeVisionControllerInterface.DataConfig.parameterData248Byte_1.commandNumber := 0;
   cmCathodeVisionControllerInterface.DataConfig.parameterData248Byte_1.cmdParameter[0..15] := 0;
   cmCathodeVisionControllerInterface.DataConfig.parameterData248Byte_1.inDataFieldbus[0..42] := 0;
   cmCathodeVisionControllerInterface.DataConfig.parameterData248Byte_2[0..61] := 0;
   cmCathodeVisionControllerInterface.DataConfig.parameterData248Byte_3[0..61] := 0;
   cmCathodeVisionControllerInterface.DataConfig.parameterData248Byte_4[0..61] := 0;
   cmCathodeVisionControllerInterface.DataConfig.parameterData248Byte_5[0..61] := 0;
   softCam.cmCathodeMainPnP1AxisX.TargetPosition := 0.0;
   softCam.cmCathodeMainPnP1AxisX.ActualPosition := 0.0;
   softCam.cmCathodeMainPnP1AxisX.UnitName := WSTRING#'';
   softCam.cmCathodeMainPnP1AxisX.error := FALSE;
   softCam.cmCathodeMainPnP1AxisX.status := 16#0000;
   softCam.cmCathodeMainPnP1AxisX.position[0..15].SetValue.Negative := 0.0;
   softCam.cmCathodeMainPnP1AxisX.position[0..15].SetValue.Postive := 0.0;
   softCam.cmCathodeMainPnP1AxisX.position[0..15].ProcessValue.Postive := 0.0;
   softCam.cmCathodeMainPnP1AxisX.position[0..15].ProcessValue.Negative := 0.0;
   softCam.cmCathodeMainPnP1AxisX.position[0..15].ProcessValue.SetPos := 0.0;
   softCam.cmCathodeMainPnP1AxisX.position[0..15].ProcessValue.inPos := FALSE;
   softCam.cmCathodeMainPnP1AxisX.position[0..15].ProcessValue.isBefore := FALSE;
   softCam.cmCathodeMainPnP1AxisX.position[0..15].ProcessValue.isAfter := FALSE;
   softCam.cmCathodeMainPnP1AxisX.position[0..15].ProcessValue.PosName := WSTRING#'';
   softCam.cmCathodeMainPnP2AxisX.TargetPosition := 0.0;
   softCam.cmCathodeMainPnP2AxisX.ActualPosition := 0.0;
   softCam.cmCathodeMainPnP2AxisX.UnitName := WSTRING#'';
   softCam.cmCathodeMainPnP2AxisX.error := FALSE;
   softCam.cmCathodeMainPnP2AxisX.status := 16#0000;
   softCam.cmCathodeMainPnP2AxisX.position[0..15].SetValue.Negative := 0.0;
   softCam.cmCathodeMainPnP2AxisX.position[0..15].SetValue.Postive := 0.0;
   softCam.cmCathodeMainPnP2AxisX.position[0..15].ProcessValue.Postive := 0.0;
   softCam.cmCathodeMainPnP2AxisX.position[0..15].ProcessValue.Negative := 0.0;
   softCam.cmCathodeMainPnP2AxisX.position[0..15].ProcessValue.SetPos := 0.0;
   softCam.cmCathodeMainPnP2AxisX.position[0..15].ProcessValue.inPos := FALSE;
   softCam.cmCathodeMainPnP2AxisX.position[0..15].ProcessValue.isBefore := FALSE;
   softCam.cmCathodeMainPnP2AxisX.position[0..15].ProcessValue.isAfter := FALSE;
   softCam.cmCathodeMainPnP2AxisX.position[0..15].ProcessValue.PosName := WSTRING#'';
   softCam.cmCathodeMainPnP1AxisY.TargetPosition := 0.0;
   softCam.cmCathodeMainPnP1AxisY.ActualPosition := 0.0;
   softCam.cmCathodeMainPnP1AxisY.UnitName := WSTRING#'';
   softCam.cmCathodeMainPnP1AxisY.error := FALSE;
   softCam.cmCathodeMainPnP1AxisY.status := 16#0000;
   softCam.cmCathodeMainPnP1AxisY.position[0..15].SetValue.Negative := 0.0;
   softCam.cmCathodeMainPnP1AxisY.position[0..15].SetValue.Postive := 0.0;
   softCam.cmCathodeMainPnP1AxisY.position[0..15].ProcessValue.Postive := 0.0;
   softCam.cmCathodeMainPnP1AxisY.position[0..15].ProcessValue.Negative := 0.0;
   softCam.cmCathodeMainPnP1AxisY.position[0..15].ProcessValue.SetPos := 0.0;
   softCam.cmCathodeMainPnP1AxisY.position[0..15].ProcessValue.inPos := FALSE;
   softCam.cmCathodeMainPnP1AxisY.position[0..15].ProcessValue.isBefore := FALSE;
   softCam.cmCathodeMainPnP1AxisY.position[0..15].ProcessValue.isAfter := FALSE;
   softCam.cmCathodeMainPnP1AxisY.position[0..15].ProcessValue.PosName := WSTRING#'';
   softCam.cmCathodeMainPnP1AxisZ.TargetPosition := 0.0;
   softCam.cmCathodeMainPnP1AxisZ.ActualPosition := 0.0;
   softCam.cmCathodeMainPnP1AxisZ.UnitName := WSTRING#'';
   softCam.cmCathodeMainPnP1AxisZ.error := FALSE;
   softCam.cmCathodeMainPnP1AxisZ.status := 16#0000;
   softCam.cmCathodeMainPnP1AxisZ.position[0..15].SetValue.Negative := 0.0;
   softCam.cmCathodeMainPnP1AxisZ.position[0..15].SetValue.Postive := 0.0;
   softCam.cmCathodeMainPnP1AxisZ.position[0..15].ProcessValue.Postive := 0.0;
   softCam.cmCathodeMainPnP1AxisZ.position[0..15].ProcessValue.Negative := 0.0;
   softCam.cmCathodeMainPnP1AxisZ.position[0..15].ProcessValue.SetPos := 0.0;
   softCam.cmCathodeMainPnP1AxisZ.position[0..15].ProcessValue.inPos := FALSE;
   softCam.cmCathodeMainPnP1AxisZ.position[0..15].ProcessValue.isBefore := FALSE;
   softCam.cmCathodeMainPnP1AxisZ.position[0..15].ProcessValue.isAfter := FALSE;
   softCam.cmCathodeMainPnP1AxisZ.position[0..15].ProcessValue.PosName := WSTRING#'';
   softCam.cmCathodeMainPnP2AxisZ.TargetPosition := 0.0;
   softCam.cmCathodeMainPnP2AxisZ.ActualPosition := 0.0;
   softCam.cmCathodeMainPnP2AxisZ.UnitName := WSTRING#'';
   softCam.cmCathodeMainPnP2AxisZ.error := FALSE;
   softCam.cmCathodeMainPnP2AxisZ.status := 16#0000;
   softCam.cmCathodeMainPnP2AxisZ.position[0..15].SetValue.Negative := 0.0;
   softCam.cmCathodeMainPnP2AxisZ.position[0..15].SetValue.Postive := 0.0;
   softCam.cmCathodeMainPnP2AxisZ.position[0..15].ProcessValue.Postive := 0.0;
   softCam.cmCathodeMainPnP2AxisZ.position[0..15].ProcessValue.Negative := 0.0;
   softCam.cmCathodeMainPnP2AxisZ.position[0..15].ProcessValue.SetPos := 0.0;
   softCam.cmCathodeMainPnP2AxisZ.position[0..15].ProcessValue.inPos := FALSE;
   softCam.cmCathodeMainPnP2AxisZ.position[0..15].ProcessValue.isBefore := FALSE;
   softCam.cmCathodeMainPnP2AxisZ.position[0..15].ProcessValue.isAfter := FALSE;
   softCam.cmCathodeMainPnP2AxisZ.position[0..15].ProcessValue.PosName := WSTRING#'';
   softCam.cmCathodeAlignTableAxisX.TargetPosition := 0.0;
   softCam.cmCathodeAlignTableAxisX.ActualPosition := 0.0;
   softCam.cmCathodeAlignTableAxisX.UnitName := WSTRING#'';
   softCam.cmCathodeAlignTableAxisX.error := FALSE;
   softCam.cmCathodeAlignTableAxisX.status := 16#0000;
   softCam.cmCathodeAlignTableAxisX.position[0..15].SetValue.Negative := 0.0;
   softCam.cmCathodeAlignTableAxisX.position[0..15].SetValue.Postive := 0.0;
   softCam.cmCathodeAlignTableAxisX.position[0..15].ProcessValue.Postive := 0.0;
   softCam.cmCathodeAlignTableAxisX.position[0..15].ProcessValue.Negative := 0.0;
   softCam.cmCathodeAlignTableAxisX.position[0..15].ProcessValue.SetPos := 0.0;
   softCam.cmCathodeAlignTableAxisX.position[0..15].ProcessValue.inPos := FALSE;
   softCam.cmCathodeAlignTableAxisX.position[0..15].ProcessValue.isBefore := FALSE;
   softCam.cmCathodeAlignTableAxisX.position[0..15].ProcessValue.isAfter := FALSE;
   softCam.cmCathodeAlignTableAxisX.position[0..15].ProcessValue.PosName := WSTRING#'';
   softCam.cmCathodeAlignTableAxisY1.TargetPosition := 0.0;
   softCam.cmCathodeAlignTableAxisY1.ActualPosition := 0.0;
   softCam.cmCathodeAlignTableAxisY1.UnitName := WSTRING#'';
   softCam.cmCathodeAlignTableAxisY1.error := FALSE;
   softCam.cmCathodeAlignTableAxisY1.status := 16#0000;
   softCam.cmCathodeAlignTableAxisY1.position[0..15].SetValue.Negative := 0.0;
   softCam.cmCathodeAlignTableAxisY1.position[0..15].SetValue.Postive := 0.0;
   softCam.cmCathodeAlignTableAxisY1.position[0..15].ProcessValue.Postive := 0.0;
   softCam.cmCathodeAlignTableAxisY1.position[0..15].ProcessValue.Negative := 0.0;
   softCam.cmCathodeAlignTableAxisY1.position[0..15].ProcessValue.SetPos := 0.0;
   softCam.cmCathodeAlignTableAxisY1.position[0..15].ProcessValue.inPos := FALSE;
   softCam.cmCathodeAlignTableAxisY1.position[0..15].ProcessValue.isBefore := FALSE;
   softCam.cmCathodeAlignTableAxisY1.position[0..15].ProcessValue.isAfter := FALSE;
   softCam.cmCathodeAlignTableAxisY1.position[0..15].ProcessValue.PosName := WSTRING#'';
   softCam.cmCathodeAlignTableAxisY2.TargetPosition := 0.0;
   softCam.cmCathodeAlignTableAxisY2.ActualPosition := 0.0;
   softCam.cmCathodeAlignTableAxisY2.UnitName := WSTRING#'';
   softCam.cmCathodeAlignTableAxisY2.error := FALSE;
   softCam.cmCathodeAlignTableAxisY2.status := 16#0000;
   softCam.cmCathodeAlignTableAxisY2.position[0..15].SetValue.Negative := 0.0;
   softCam.cmCathodeAlignTableAxisY2.position[0..15].SetValue.Postive := 0.0;
   softCam.cmCathodeAlignTableAxisY2.position[0..15].ProcessValue.Postive := 0.0;
   softCam.cmCathodeAlignTableAxisY2.position[0..15].ProcessValue.Negative := 0.0;
   softCam.cmCathodeAlignTableAxisY2.position[0..15].ProcessValue.SetPos := 0.0;
   softCam.cmCathodeAlignTableAxisY2.position[0..15].ProcessValue.inPos := FALSE;
   softCam.cmCathodeAlignTableAxisY2.position[0..15].ProcessValue.isBefore := FALSE;
   softCam.cmCathodeAlignTableAxisY2.position[0..15].ProcessValue.isAfter := FALSE;
   softCam.cmCathodeAlignTableAxisY2.position[0..15].ProcessValue.PosName := WSTRING#'';
END_DATA_BLOCK
